FUNCTION "FC_ArbiterMech" : USInt
{ S7_Optimized_Access := 'TRUE' }
VERSION : 0.1
// Повертає RejectCode:
//   0 = ARB_OK (успішно)
//   1 = ARB_LOCAL_MANUAL (локальний режим активний)
//   2 = ARB_OWNER_BUSY (зайнято іншим власником)
//   3 = ARB_WRONG_STATUS (неправильний статус для операції)
//   4 = ARB_SLOT_INVALID (невалідний слот/немапований)
//   5 = ARB_CMD_BLOCKED (команда заблокована, напр. CMD_SET_FORCE)
//   6 = ARB_CMD_INVALID (невалідна команда, CMD_NONE)
//
// Meta-команди (розпізнаються автоматично):
//   CMD_RELEASE_OWNER - звільняє власника
//   CMD_SET_OWNER_SCADA - тільки захоплює власника (без виконання команди)
   VAR_INPUT
      OwnerReq : USInt;   // ID запитувача (DB_Const.OWNER_*)
      OwnerReqId : UInt;   // Додатковий ID (наприклад, Route ID)
      ReqCmd : USInt;   // Команда (DB_Const.CMD_*)
      ReqParam1 : Int;   // Параметр команди
   END_VAR

   VAR_IN_OUT
      M : "UDT_BaseMechanism";   // Структура механізму
   END_VAR

   VAR_TEMP
      rejectCode : USInt;   // Код помилки (0 = OK)
      okOwner : Bool;
   END_VAR


BEGIN


	// =========================================================
	// ПЕРЕВІРКА 1: Валідація слоту
	// =========================================================
	IF (#M.SlotId > "MECHS_COUNT") OR (#M.DeviceType = "TYPE_NONE") OR (#M.TypedIndex = UINT#16#FFFF) THEN
	    #FC_ArbiterMech := "ARB_SLOT_INVALID";

	    RETURN;
	END_IF;

	// =========================================================
	// ПЕРЕВІРКА 2: Локальний режим (блокує всі операції)
	// =========================================================
	IF "GlobalLocalManual" OR #M.LocalManual THEN
	    #FC_ArbiterMech := "ARB_LOCAL_MANUAL";

	    RETURN;
	END_IF;

	// =========================================================
	// META-КОМАНДА: CMD_RELEASE_OWNER (звільнити власника)
	// =========================================================
	IF #ReqCmd = "CMD_RELEASE_OWNER" THEN // CMD_RELEASE_OWNER

	    // Перевірка: чи запитувач є поточним власником?
	    #okOwner := (#M.OwnerCur = #OwnerReq) AND (#M.OwnerCurId = #OwnerReqId);
	    IF NOT #okOwner THEN
	        #FC_ArbiterMech := "ARB_OWNER_BUSY";

	        RETURN;
	    END_IF;

	    // Перевірка: дозволяємо скинути власника в IDLE, FAULT або STOPPING
	    IF NOT (#M.Status = "STS_IDLE" OR #M.Status = "STS_FAULT" OR #M.Status = "STS_STOPPING") THEN
	        #FC_ArbiterMech := "ARB_WRONG_STATUS";

	        RETURN;
	    END_IF;

	    // Звільнення власника
	    #M.OwnerCur := "OWNER_NONE";
	    #M.OwnerCurId := 0;
	    #M.LastCmd := "CMD_RELEASE_OWNER";
	    #FC_ArbiterMech := "ARB_OK";

	    RETURN;

	END_IF;

	// =========================================================
	// META-КОМАНДА: CMD_SET_OWNER_SCADA (тільки захопити)
	// =========================================================
	IF #ReqCmd = "CMD_SET_OWNER_SCADA" THEN

	    // Захоплення owner (якщо він вільний)
	    IF (#M.OwnerCur = "OWNER_NONE") AND (#OwnerReq <> "OWNER_NONE") THEN
	        // Дозволяємо захоплення в IDLE, FAULT або STOPPING
	        // STS_STOPPING додано бо маршрут може перезапускатись після зупинки
	        IF (#M.Status = "STS_IDLE" OR #M.Status = "STS_FAULT" OR #M.Status = "STS_STOPPING") THEN
	            #M.OwnerCur := #OwnerReq;
	            #M.OwnerCurId := #OwnerReqId;
	            #M.LastCmd := "CMD_SET_OWNER_SCADA";
	            #FC_ArbiterMech := "ARB_OK";

	        ELSE
	            #FC_ArbiterMech := "ARB_WRONG_STATUS";

	        END_IF;
	    ELSE
	        // Перевірка: чи запитувач вже є власником?
	        #okOwner := (#M.OwnerCur = #OwnerReq) AND (#M.OwnerCurId = #OwnerReqId);
	        IF #okOwner THEN
	            #FC_ArbiterMech := "ARB_OK";

	        ELSE
	            #FC_ArbiterMech := "ARB_OWNER_BUSY";

	        END_IF;
	    END_IF;
	    RETURN;

	END_IF;

	// =========================================================
	// ЗВИЧАЙНІ КОМАНДИ (захоплення + виконання)
	// =========================================================

	// Перевірка: CMD_NONE заборонено
	IF #ReqCmd = "CMD_NONE" THEN
	    #FC_ArbiterMech := "ARB_CMD_INVALID";

	    RETURN;
	END_IF;

	// Захоплення owner (якщо він вільний)
	IF (#M.OwnerCur = "OWNER_NONE") AND (#OwnerReq <> "OWNER_NONE") THEN
	    // Дозволяємо захоплення тільки в IDLE (0) або FAULT
	    IF (#M.Status = "STS_IDLE" OR #M.Status = "STS_FAULT") THEN
	        #M.OwnerCur := #OwnerReq;
	        #M.OwnerCurId := #OwnerReqId;
	    ELSE
	        #FC_ArbiterMech := "ARB_WRONG_STATUS";

	        RETURN;
	    END_IF;
	END_IF;

	// Перевірка: чи запитувач є власником?
	#okOwner := (#M.OwnerCur = #OwnerReq) AND (#M.OwnerCurId = #OwnerReqId);
	IF NOT #okOwner THEN
	    #FC_ArbiterMech := "ARB_OWNER_BUSY";

	    RETURN;
	END_IF;

	// Виконання команди
	#M.Cmd := #ReqCmd;
	#M.CmdParam1 := #ReqParam1;

	#FC_ArbiterMech := "ARB_OK";

END_FUNCTION

